// TIA Portal V20 export
FUNCTION_BLOCK "FB_Position"   // FB38, SCL
{ S7_Optimized_Access := 'TRUE' }
// stored: MemoryReserve 100, SetENOAutomatically false
   VAR_INPUT
      iCondPartInSh1 : Bool;
      iCondBwInSh1 : Bool;
      iCondPartInSh2 : Bool;
      iCondBwInSh2 : Bool;
      iCondPartPresCtrlInSh1 : Bool;
      iCondBWPresCtrlInSh1 : Bool;
      iCondPartPresCtrlInSh2 : Bool;
      iCondBWPresCtrlInSh2 : Bool;
      iCondPartPresCtrlOutSh1 : Bool;
      iCondPartPresCtrlOutSh2 : Bool;
      iUndrilledPartPresence : Bool;
      iDrilledPartPresence : Bool;
      iUndrilledBWPresence : Bool;
      iCloseReqLoadGripperSh1 : Bool;
      iCloseReqLoadGripperSh2 : Bool;
      iCloseReqFixture : Bool;
      iDrilling_Finished : Bool;
      iCloseReqUnloadGripper : Bool;
      iOpenReqUnloadGripperSh1 : Bool;
      iOpenReqUnloadGripperSh2 : Bool;
      iCondPartOutSh1 : Bool;
      iCondBwOutSh1 : Bool;
      iCondPartOutSh2 : Bool;
      iCondBwOutSh2 : Bool;
   END_VAR
   VAR RETAIN
      sShuttle1 : "UDT_PartPosition";
      sShuttle2 { S7_SetPoint := 'True'} : "UDT_PartPosition";
      sGripper { S7_SetPoint := 'True'} : "UDT_PartPosition";
      sFixture { S7_SetPoint := 'True'} : "UDT_PartPosition";
   END_VAR
   VAR
      sRT_PartInSh1 : R_TRIG;
      sRT_BwInSh1 : R_TRIG;
      sRT_PartInSh2 : R_TRIG;
      sRT_BwInSh2 : R_TRIG;
      sRT_PartPresenceInSh1 { S7_SetPoint := 'True'} : R_TRIG;
      sRT_BWPresenceInSh1 { S7_SetPoint := 'True'} : R_TRIG;
      sRT_PartPresenceInSh2 { S7_SetPoint := 'True'} : R_TRIG;
      sRT_BWPresenceInSh2 { S7_SetPoint := 'True'} : R_TRIG;
      sRT_PartPresenceOutSh1 { S7_SetPoint := 'True'} : R_TRIG;
      sRT_PartPresenceOutSh2 { S7_SetPoint := 'True'} : R_TRIG;
      sRT_CloseLoadGripperSh1 : R_TRIG;
      sRT_CloseLoadGripperSh2 : R_TRIG;
      sRT_CloseFixture { S7_SetPoint := 'True'} : R_TRIG;
      sRT_Drilling_Finished { S7_SetPoint := 'True'} : R_TRIG;
      sRT_CloseUnloadGripper { S7_SetPoint := 'True'} : R_TRIG;
      sRT_OpenUnloadGripperSh1 { S7_SetPoint := 'True'} : R_TRIG;
      sRT_OpenUnloadGripperSh2 { S7_SetPoint := 'True'} : R_TRIG;
      sRT_PartOutSh1 : R_TRIG;
      sRT_BwOutSh1 : R_TRIG;
      sRT_PartOutSh2 : R_TRIG;
      sRT_BwOutSh2 : R_TRIG;
      sMachineEmpty { S7_SetPoint := 'True'} : Bool;
      sShuttle1Empty { S7_SetPoint := 'True'} : Bool;
      sShuttle2Empty { S7_SetPoint := 'True'} : Bool;
      sGripperEmpty { S7_SetPoint := 'True'} : Bool;
      sFixtureEmpty { S7_SetPoint := 'True'} : Bool;
      sPartNumber : Struct
         Shuttle1 : Int;
         Shuttle2 : Int;
         Gripper : Int;
         Fixture : Int;
         Total : Int;
      END_STRUCT;
      sEmptyPosition { S7_SetPoint := 'True'} : "UDT_EmptyPosition";
      sTON_PartPresenceOutSh1 { S7_SetPoint := 'True'} : TON_TIME;
      sTON_PartPresenceOutSh2 { S7_SetPoint := 'True'} : TON_TIME;
   END_VAR
BEGIN
   REGION Description header 
       //==================================================================================
       // POSALUX Swiss SA / (C) Copyright 2025
       //----------------------------------------------------------------------------------
       // Title: FB_Position
       // Comment/Function: 
       // Author: Fabien WALDT
       // Engineering: TIA Portal v17
       //----------------------------------------------------------------------------------
       // Change log table:
       // Version  | Date     | Expert in charge | Changes applied
       // ---------|----------|------------------|-----------------------------------------
       // 00.00.01 | 20250423 | WFA              | First released version
       // =================================================================================
   END_REGION

   REGION Input Part/BW Shuttle 1 (Loading)
       // Part
       #sRT_PartInSh1(CLK := #iCondPartInSh1);
       IF #sRT_PartInSh1.Q AND NOT "LBP_ModeGroup".E_JOG THEN
           #sShuttle1.Undrilled.Presence.Part := TRUE;
       END_IF;

       // BW
       #sRT_BwInSh1(CLK := #iCondBwInSh1);
       IF #sRT_BwInSh1.Q AND NOT "LBP_ModeGroup".E_JOG THEN
           #sShuttle1.Undrilled.Presence.BW := TRUE;
       END_IF;
   END_REGION

   REGION Input Part/BW Shuttle 2 (Loading)
       // Part
       #sRT_PartInSh2(CLK := #iCondPartInSh2);
       IF #sRT_PartInSh2.Q AND NOT "LBP_ModeGroup".E_JOG THEN
           #sShuttle2.Undrilled.Presence.Part := TRUE;
       END_IF;

       // BW
       #sRT_BwInSh2(CLK := #iCondBwInSh2);
       IF #sRT_BwInSh2.Q AND NOT "LBP_ModeGroup".E_JOG THEN
           #sShuttle2.Undrilled.Presence.BW := TRUE;
       END_IF;
   END_REGION

   REGION Input Part/BW Shuttle 1 (Control IN)
       // Part
       #sRT_PartPresenceInSh1(CLK := #iCondPartPresCtrlInSh1);
       IF #sRT_PartPresenceInSh1.Q AND NOT "LBP_ModeGroup".E_JOG THEN
           #sShuttle1.Undrilled.Presence.Part := #iUndrilledPartPresence;
           #sShuttle1.Drilled.Presence.Part := #iDrilledPartPresence;
       END_IF;

      // BW
       #sRT_BWPresenceInSh1(CLK := #iCondBWPresCtrlInSh1);
       IF #sRT_BWPresenceInSh1.Q AND NOT "LBP_ModeGroup".E_JOG THEN
           #sShuttle1.Undrilled.Presence.BW := #iUndrilledBWPresence;
       END_IF;
   END_REGION

   REGION Input Part/BW Shuttle 2 (Control IN)
       // Part
       #sRT_PartPresenceInSh2(CLK := #iCondPartPresCtrlInSh2);

       IF #sRT_PartPresenceInSh2.Q AND NOT "LBP_ModeGroup".E_JOG THEN
           #sShuttle2.Undrilled.Presence.Part := #iUndrilledPartPresence;
           #sShuttle2.Drilled.Presence.Part := #iDrilledPartPresence;
       END_IF;

       // BW
       #sRT_BWPresenceInSh2(CLK := #iCondBWPresCtrlInSh2);

       IF #sRT_BWPresenceInSh2.Q AND NOT "LBP_ModeGroup".E_JOG THEN
           #sShuttle2.Undrilled.Presence.BW := #iUndrilledBWPresence;
       END_IF;
   END_REGION

   REGION Transfert Shuttle 1/2 to Gripper U
       #sRT_CloseLoadGripperSh1(CLK := #iCloseReqLoadGripperSh1);
       #sRT_CloseLoadGripperSh2(CLK := #iCloseReqLoadGripperSh2);

       IF #sRT_CloseLoadGripperSh1.Q AND NOT "LBP_ModeGroup".E_JOG THEN
           #sGripper.Undrilled := #sShuttle1.Undrilled;
           #sShuttle1.Undrilled := #sEmptyPosition;
       ELSIF #sRT_CloseLoadGripperSh2.Q AND NOT "LBP_ModeGroup".E_JOG THEN
           #sGripper.Undrilled := #sShuttle2.Undrilled;
           #sShuttle2.Undrilled := #sEmptyPosition;
       END_IF;
   END_REGION

   REGION Transfert Gripper U to Fixture
       #sRT_CloseFixture(CLK := #iCloseReqFixture);

       IF #sRT_CloseFixture.Q AND NOT "LBP_ModeGroup".E_JOG THEN
           #sFixture.Undrilled :=  #sGripper.Undrilled;
           #sGripper.Undrilled := #sEmptyPosition;
       END_IF;
   END_REGION

   REGION Transfert Fixture Undrilled to Fixture Drilled
       #sRT_Drilling_Finished(CLK := #iDrilling_Finished);

       IF #sRT_Drilling_Finished.Q AND NOT "LBP_ModeGroup".E_JOG THEN
       #sFixture.Drilled := #sFixture.Undrilled;
           #sFixture.Undrilled := #sEmptyPosition;
       END_IF;
   END_REGION

   REGION Transfert Fixture to Gripper D
       #sRT_CloseUnloadGripper(CLK := #iCloseReqUnloadGripper);

       IF #sRT_CloseUnloadGripper.Q AND NOT "LBP_ModeGroup".E_JOG THEN
           #sGripper.Drilled := #sFixture.Drilled;
           #sFixture.Drilled := #sEmptyPosition;
       END_IF;
   END_REGION

   REGION Transfert Gripper D to Shuttle 1/2
       #sRT_OpenUnloadGripperSh1(CLK := #iOpenReqUnloadGripperSh1);
       #sRT_OpenUnloadGripperSh2(CLK := #iOpenReqUnloadGripperSh2);

       IF #sRT_OpenUnloadGripperSh1.Q AND NOT "LBP_ModeGroup".E_JOG THEN
           #sShuttle1.Drilled := #sGripper.Drilled;
           #sGripper.Drilled := #sEmptyPosition;
       ELSIF #sRT_OpenUnloadGripperSh2.Q AND NOT "LBP_ModeGroup".E_JOG THEN
           #sShuttle2.Drilled := #sGripper.Drilled;
           #sGripper.Drilled := #sEmptyPosition;
       END_IF;
   END_REGION

   REGION Output Part/BW Shuttle 1 (Unloading)
       // Part
       #sRT_PartOutSh1(CLK := #iCondPartOutSh1);
       IF #sRT_PartOutSh1.Q AND NOT "LBP_ModeGroup".E_JOG THEN
           #sShuttle1.Drilled.Presence.Part := FALSE;
       END_IF;

       // BW
       #sRT_BwOutSh1(CLK := #iCondBwOutSh1);
       IF #sRT_BwOutSh1.Q AND NOT "LBP_ModeGroup".E_JOG THEN
           #sShuttle1.Drilled.Presence.BW := FALSE;
       END_IF;
   END_REGION

   REGION Output Part/BW Shuttle 2 (Unloading)
       // Part
       #sRT_PartOutSh2(CLK := #iCondPartOutSh2);
       IF #sRT_PartOutSh2.Q AND NOT "LBP_ModeGroup".E_JOG THEN
           #sShuttle2.Drilled.Presence.Part := FALSE;
       END_IF;

       // BW
       #sRT_BwOutSh2(CLK := #iCondBwOutSh2);
       IF #sRT_BwOutSh2.Q AND NOT "LBP_ModeGroup".E_JOG THEN
           #sShuttle2.Drilled.Presence.BW := FALSE;
       END_IF;
   END_REGION

   REGION Output Part/BW Shuttle 1 (Control OUT)
       // Part
       #sTON_PartPresenceOutSh1(IN := #iCondPartPresCtrlOutSh1,
                                PT := t#100ms);

       #sRT_PartPresenceOutSh1(CLK := #sTON_PartPresenceOutSh1.Q);

       IF #sRT_PartPresenceOutSh1.Q AND NOT "LBP_ModeGroup".E_JOG THEN
           #sShuttle1.Undrilled.Presence.Part := #iUndrilledPartPresence;
           #sShuttle1.Drilled.Presence.Part := #iDrilledPartPresence;
       END_IF;

       // BW - No BW Control at output
   END_REGION

   REGION Output Part/BW Shuttle 2 (Control OUT)
       // Part
       #sTON_PartPresenceOutSh2(IN := #iCondPartPresCtrlOutSh2,
                                PT := t#100ms);

       #sRT_PartPresenceOutSh2(CLK := #iCondPartPresCtrlOutSh2);

       IF #sRT_PartPresenceOutSh2.Q AND NOT "LBP_ModeGroup".E_JOG THEN
           #sShuttle2.Undrilled.Presence.Part := #iUndrilledPartPresence;
           #sShuttle2.Drilled.Presence.Part := #iDrilledPartPresence;
       END_IF;

       // BW - No BW Control at output
   END_REGION

   REGION Machine states
       // Shuttle 1 Empty
       #sShuttle1Empty :=
       NOT #sShuttle1.Undrilled.Presence.Part
       AND NOT #sShuttle1.Undrilled.Presence.BW
       AND NOT #sShuttle1.Drilled.Presence.Part
       AND NOT #sShuttle1.Drilled.Presence.BW;

       // Shuttle 2 Empty
       #sShuttle2Empty :=
       NOT #sShuttle2.Undrilled.Presence.Part
       AND NOT #sShuttle2.Undrilled.Presence.BW
       AND NOT #sShuttle2.Drilled.Presence.Part
       AND NOT #sShuttle2.Drilled.Presence.BW;

       // Gripper Empty
       #sGripperEmpty :=
       NOT #sGripper.Undrilled.Presence.Part
       AND NOT #sGripper.Undrilled.Presence.BW
       AND NOT #sGripper.Drilled.Presence.Part
       AND NOT #sGripper.Drilled.Presence.BW;

       // Fixture Empty
       #sFixtureEmpty :=
       NOT #sFixture.Undrilled.Presence.Part
       AND NOT #sFixture.Undrilled.Presence.BW
       AND NOT #sFixture.Drilled.Presence.Part
       AND NOT #sFixture.Drilled.Presence.BW;

       // Machine Empty
       #sMachineEmpty := #sShuttle1Empty
       AND #sShuttle2Empty
       AND #sGripperEmpty
       AND #sFixtureEmpty;
   END_REGION

   REGION Part in Machine
       // Shuttle 1
       #sPartNumber.Shuttle1 := 0;
       IF #sShuttle1.Undrilled.Presence.Part AND #sShuttle1.Drilled.Presence.Part THEN
           #sPartNumber.Shuttle1 := 2;
       ELSIF #sShuttle1.Undrilled.Presence.Part XOR #sShuttle1.Drilled.Presence.Part THEN
           #sPartNumber.Shuttle1 := 1;
       END_IF;

       // Shuttle 2
       #sPartNumber.Shuttle2 := 0;
       IF #sShuttle2.Undrilled.Presence.Part AND #sShuttle2.Drilled.Presence.Part THEN
           #sPartNumber.Shuttle2 := 2;
       ELSIF #sShuttle2.Undrilled.Presence.Part XOR #sShuttle2.Drilled.Presence.Part THEN
           #sPartNumber.Shuttle2 := 1;
       END_IF;

       // Gripper
       #sPartNumber.Gripper := 0;
       IF #sGripper.Undrilled.Presence.Part AND #sGripper.Drilled.Presence.Part THEN
           #sPartNumber.Gripper := 2;
       ELSIF #sGripper.Undrilled.Presence.Part XOR #sGripper.Drilled.Presence.Part THEN
           #sPartNumber.Gripper := 1;
       END_IF;

       // Fixture
       #sPartNumber.Fixture := 0;
       IF #sFixture.Undrilled.Presence.Part OR #sFixture.Drilled.Presence.Part THEN
           #sPartNumber.Fixture := 1;
       END_IF;

       // Total
       #sPartNumber.Total := #sPartNumber.Shuttle1 + #sPartNumber.Shuttle2 + #sPartNumber.Gripper + #sPartNumber.Fixture;
   END_REGION
END_FUNCTION_BLOCK
